// TIA Portal V16 export
// export: Created 2024-09-05T17:36:33.426115Z, ExportSetting WithDefaults, DisplayName Totally Integrated Automation Portal, DisplayVersion V16 Update 6, DisplayName TIA Portal Version Control Interface, DisplayVersion V16 Update 2, DisplayName TIA Portal Openness, DisplayVersion V16 Update 6, DisplayName STEP 7 Professional, DisplayVersion V16 Update 6, DisplayName STEP 7 Safety, DisplayVersion V16, DisplayName WinCC Advanced, DisplayVersion V16 Update 6
VAR_GLOBAL   // PLC tag table "Electronic key system"
   iEksDiagnosticByte AT %IB400 : Byte;   // EKS: Diagnostic byte
   iEksKeyInserted AT %I400.1 : Bool;   // EKS: Key is inserted in reader
   iEksLevel AT %IB401 : Byte;   // EKS: Level
   iEksEmployeeID_1 AT %IB421 : Byte;   // EKS: Employee ID 1
   iEksEmployeeID_2 AT %IB422 : Byte;   // EKS: Employee ID 2
   iEksEmployeeID_3 AT %IB423 : Byte;   // EKS: Employee ID 3
   iEksEmployeeID_4 AT %IB424 : Byte;   // EKS: Employee ID 4
   iEksKeyID_1 AT %IB517 : Byte;   // EKS: Key ID 1
   iEksKeyID_2 AT %IB518 : Byte;   // EKS: Key ID 2
   iEksKeyID_3 AT %IB519 : Byte;   // EKS: Key ID 3
   iEksKeyID_4 AT %IB520 : Byte;   // EKS: Key ID 4
   iEksKeyID_5 AT %IB521 : Byte;   // EKS: Key ID 5
   iEksKeyID_6 AT %IB522 : Byte;   // EKS: Key ID 6
   iEksKeyID_7 AT %IB523 : Byte;   // EKS: Key ID 7
   iEksKeyID_8 AT %IB524 : Byte;   // EKS: Key ID 8
END_VAR
